// Mitsubishi GX Works2 project: SmartFarmModbusTempDx   PLC: FX3U/FX3UC

PROGRAM MAIN
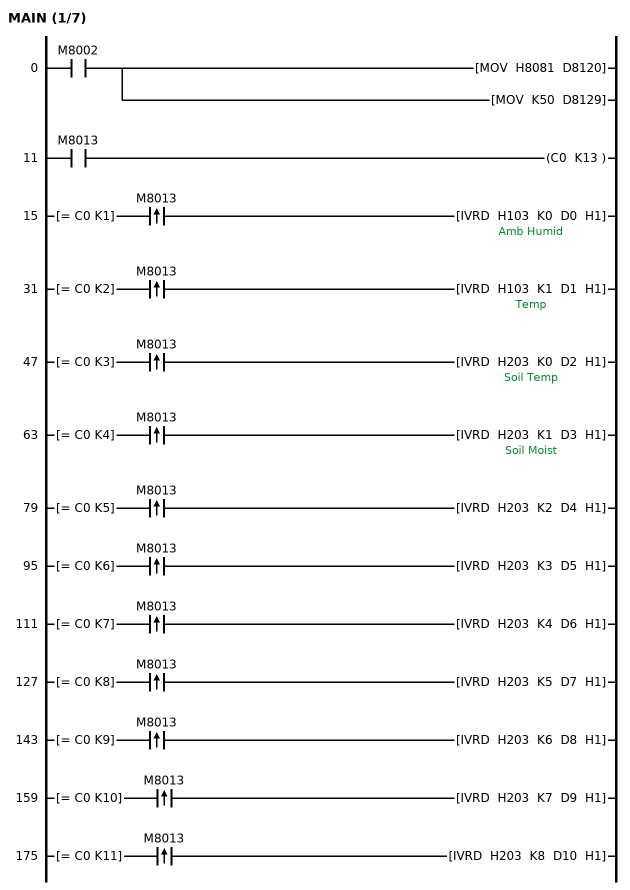
0     LD      M8002
      MOV     H8081 D8120
      MOV     K50 D8129
11    LD      M8013
      OUT     C0 K13
15    LD=     C0 K1
      ANDP    M8013
      IVRD    H103 K0 D0 H1  ; Amb Humid
31    LD=     C0 K2
      ANDP    M8013
      IVRD    H103 K1 D1 H1  ; Temp
47    LD=     C0 K3
      ANDP    M8013
      IVRD    H203 K0 D2 H1  ; Soil Temp
63    LD=     C0 K4
      ANDP    M8013
      IVRD    H203 K1 D3 H1  ; Soil Moist
79    LD=     C0 K5
      ANDP    M8013
      IVRD    H203 K2 D4 H1
95    LD=     C0 K6
      ANDP    M8013
      IVRD    H203 K3 D5 H1
111   LD=     C0 K7
      ANDP    M8013
      IVRD    H203 K4 D6 H1
127   LD=     C0 K8
      ANDP    M8013
      IVRD    H203 K5 D7 H1
143   LD=     C0 K9
      ANDP    M8013
      IVRD    H203 K6 D8 H1
159   LD=     C0 K10
      ANDP    M8013
      IVRD    H203 K7 D9 H1
175   LD=     C0 K11
      ANDP    M8013
      IVRD    H203 K8 D10 H1
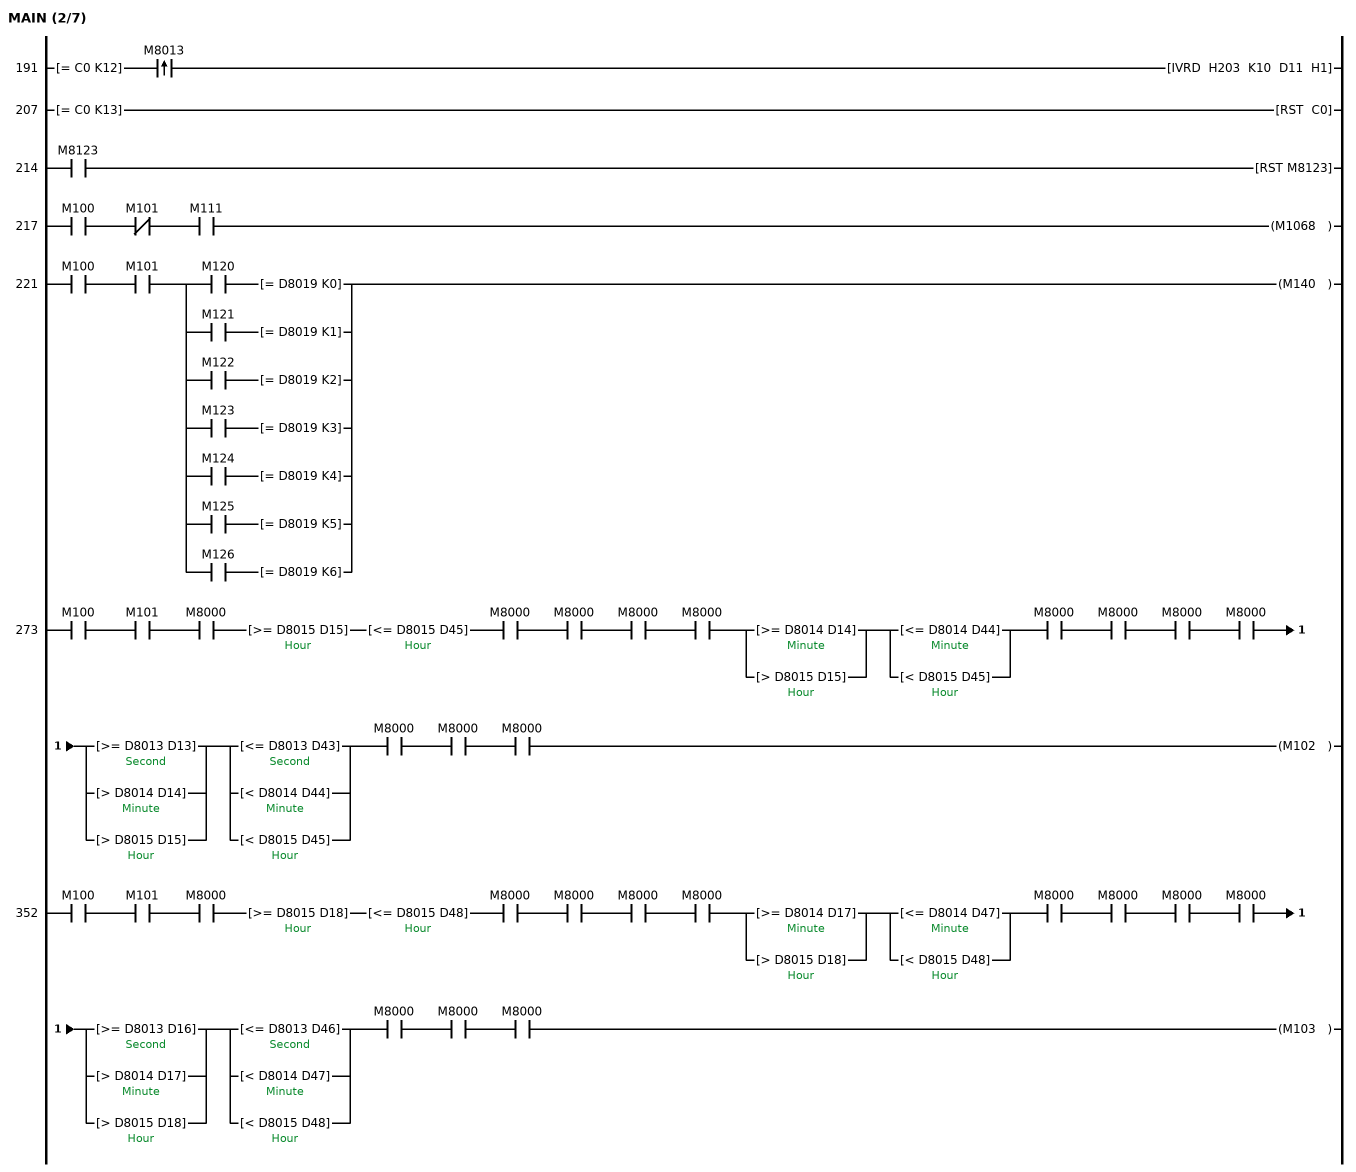
191   LD=     C0 K12
      ANDP    M8013
      IVRD    H203 K10 D11 H1
207   LD=     C0 K13
      RST     C0
214   LD      M8123
      RST     M8123
217   LD      M100
      ANI     M101
      AND     M111
      OUT     M1068
221   LD      M100
      AND     M101
      LD      M120
      AND=    D8019 K0
      LD      M121
      AND=    D8019 K1
      ORB
      LD      M122
      AND=    D8019 K2
      ORB
      LD      M123
      AND=    D8019 K3
      ORB
      LD      M124
      AND=    D8019 K4
      ORB
      LD      M125
      AND=    D8019 K5
      ORB
      LD      M126
      AND=    D8019 K6
      ORB
      ANB
      OUT     M140
273   LD      M100
      AND     M101
      AND     M8000
      AND>=   D8015 D15  ; Hour
      AND<=   D8015 D45  ; Hour
      AND     M8000
      AND     M8000
      AND     M8000
      AND     M8000
      LD>=    D8014 D14  ; Minute
      OR>     D8015 D15  ; Hour
      ANB
      LD<=    D8014 D44  ; Minute
      OR<     D8015 D45  ; Hour
      ANB
      AND     M8000
      AND     M8000
      AND     M8000
      AND     M8000
      LD>=    D8013 D13  ; Second
      OR>     D8014 D14  ; Minute
      OR>     D8015 D15  ; Hour
      ANB
      LD<=    D8013 D43  ; Second
      OR<     D8014 D44  ; Minute
      OR<     D8015 D45  ; Hour
      ANB
      AND     M8000
      AND     M8000
      AND     M8000
      OUT     M102
352   LD      M100
      AND     M101
      AND     M8000
      AND>=   D8015 D18  ; Hour
      AND<=   D8015 D48  ; Hour
      AND     M8000
      AND     M8000
      AND     M8000
      AND     M8000
      LD>=    D8014 D17  ; Minute
      OR>     D8015 D18  ; Hour
      ANB
      LD<=    D8014 D47  ; Minute
      OR<     D8015 D48  ; Hour
      ANB
      AND     M8000
      AND     M8000
      AND     M8000
      AND     M8000
      LD>=    D8013 D16  ; Second
      OR>     D8014 D17  ; Minute
      OR>     D8015 D18  ; Hour
      ANB
      LD<=    D8013 D46  ; Second
      OR<     D8014 D47  ; Minute
      OR<     D8015 D48  ; Hour
      ANB
      AND     M8000
      AND     M8000
      AND     M8000
      OUT     M103
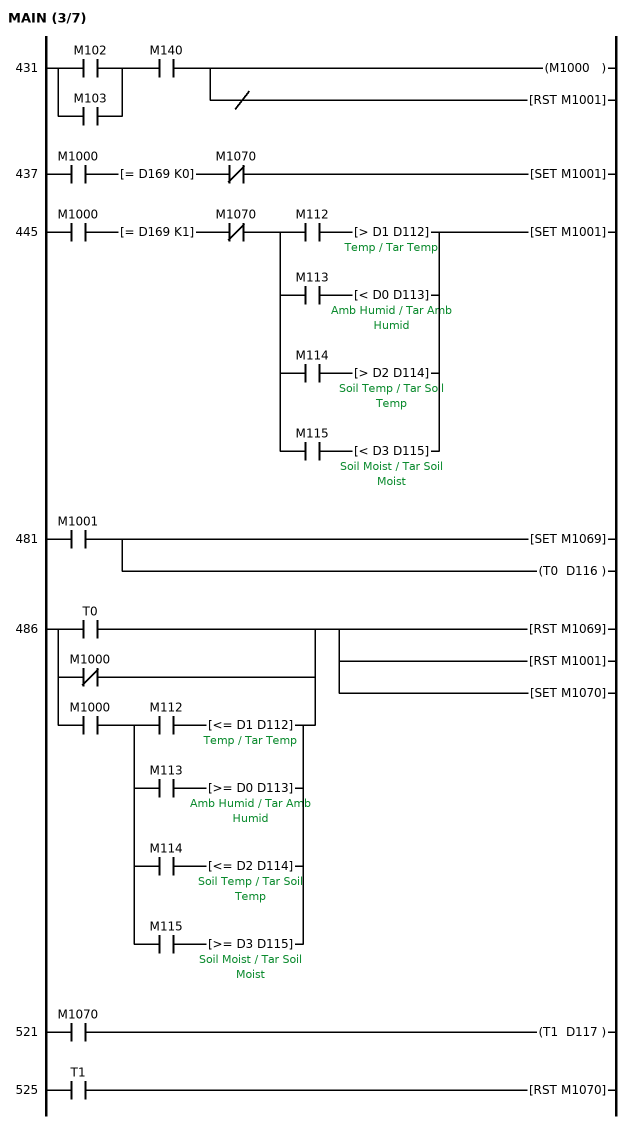
431   LD      M102
      OR      M103
      AND     M140
      OUT     M1000
      INV
      RST     M1001
437   LD      M1000
      AND=    D169 K0
      ANI     M1070
      SET     M1001
445   LD      M1000
      AND=    D169 K1
      ANI     M1070
      LD      M112
      AND>    D1 D112  ; Temp / Tar Temp
      LD      M113
      AND<    D0 D113  ; Amb Humid / Tar Amb Humid
      ORB
      LD      M114
      AND>    D2 D114  ; Soil Temp / Tar Soil Temp
      ORB
      LD      M115
      AND<    D3 D115  ; Soil Moist / Tar Soil Moist
      ORB
      ANB
      SET     M1001
481   LD      M1001
      SET     M1069
      OUT     T0 D116
486   LD      T0
      ORI     M1000
      LD      M1000
      LD      M112
      AND<=   D1 D112  ; Temp / Tar Temp
      LD      M113
      AND>=   D0 D113  ; Amb Humid / Tar Amb Humid
      ORB
      LD      M114
      AND<=   D2 D114  ; Soil Temp / Tar Soil Temp
      ORB
      LD      M115
      AND>=   D3 D115  ; Soil Moist / Tar Soil Moist
      ORB
      ANB
      ORB
      RST     M1069
      RST     M1001
      SET     M1070
521   LD      M1070
      OUT     T1 D117
525   LD      T1
      RST     M1070
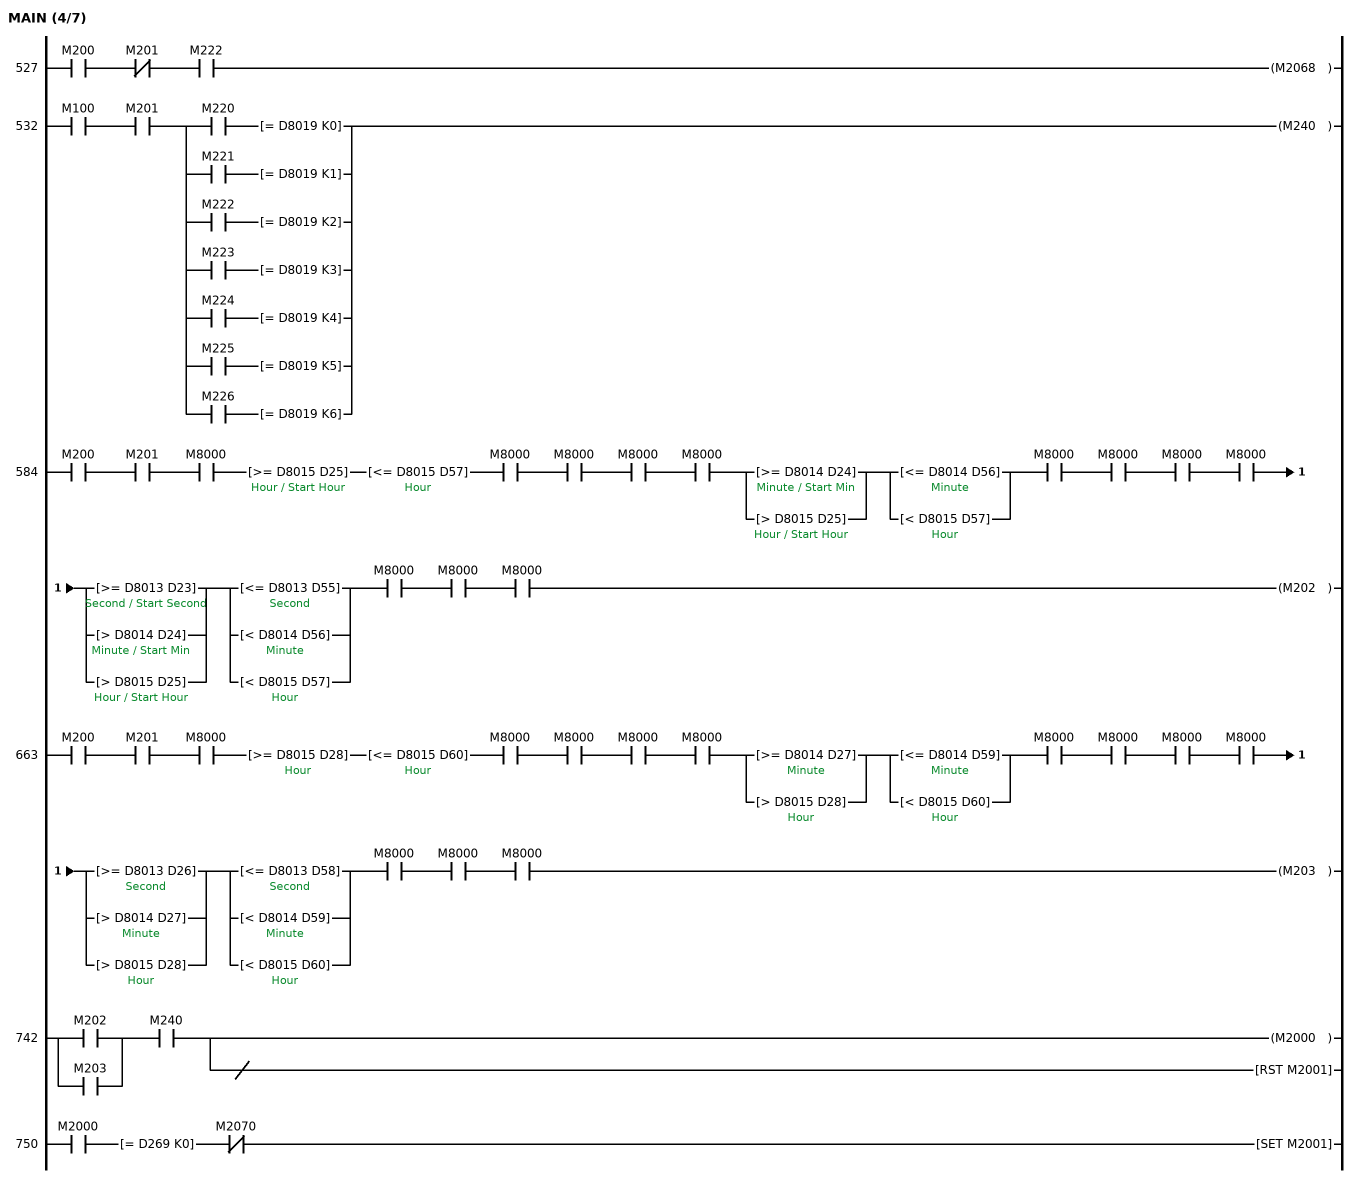
527   LD      M200
      ANI     M201
      AND     M222
      OUT     M2068
532   LD      M100
      AND     M201
      LD      M220
      AND=    D8019 K0
      LD      M221
      AND=    D8019 K1
      ORB
      LD      M222
      AND=    D8019 K2
      ORB
      LD      M223
      AND=    D8019 K3
      ORB
      LD      M224
      AND=    D8019 K4
      ORB
      LD      M225
      AND=    D8019 K5
      ORB
      LD      M226
      AND=    D8019 K6
      ORB
      ANB
      OUT     M240
584   LD      M200
      AND     M201
      AND     M8000
      AND>=   D8015 D25  ; Hour / Start Hour
      AND<=   D8015 D57  ; Hour
      AND     M8000
      AND     M8000
      AND     M8000
      AND     M8000
      LD>=    D8014 D24  ; Minute / Start Min
      OR>     D8015 D25  ; Hour / Start Hour
      ANB
      LD<=    D8014 D56  ; Minute
      OR<     D8015 D57  ; Hour
      ANB
      AND     M8000
      AND     M8000
      AND     M8000
      AND     M8000
      LD>=    D8013 D23  ; Second / Start Second
      OR>     D8014 D24  ; Minute / Start Min
      OR>     D8015 D25  ; Hour / Start Hour
      ANB
      LD<=    D8013 D55  ; Second
      OR<     D8014 D56  ; Minute
      OR<     D8015 D57  ; Hour
      ANB
      AND     M8000
      AND     M8000
      AND     M8000
      OUT     M202
663   LD      M200
      AND     M201
      AND     M8000
      AND>=   D8015 D28  ; Hour
      AND<=   D8015 D60  ; Hour
      AND     M8000
      AND     M8000
      AND     M8000
      AND     M8000
      LD>=    D8014 D27  ; Minute
      OR>     D8015 D28  ; Hour
      ANB
      LD<=    D8014 D59  ; Minute
      OR<     D8015 D60  ; Hour
      ANB
      AND     M8000
      AND     M8000
      AND     M8000
      AND     M8000
      LD>=    D8013 D26  ; Second
      OR>     D8014 D27  ; Minute
      OR>     D8015 D28  ; Hour
      ANB
      LD<=    D8013 D58  ; Second
      OR<     D8014 D59  ; Minute
      OR<     D8015 D60  ; Hour
      ANB
      AND     M8000
      AND     M8000
      AND     M8000
      OUT     M203
742   LD      M202
      OR      M203
      AND     M240
      OUT     M2000
      INV
      RST     M2001
750   LD      M2000
      AND=    D269 K0
      ANI     M2070
      SET     M2001
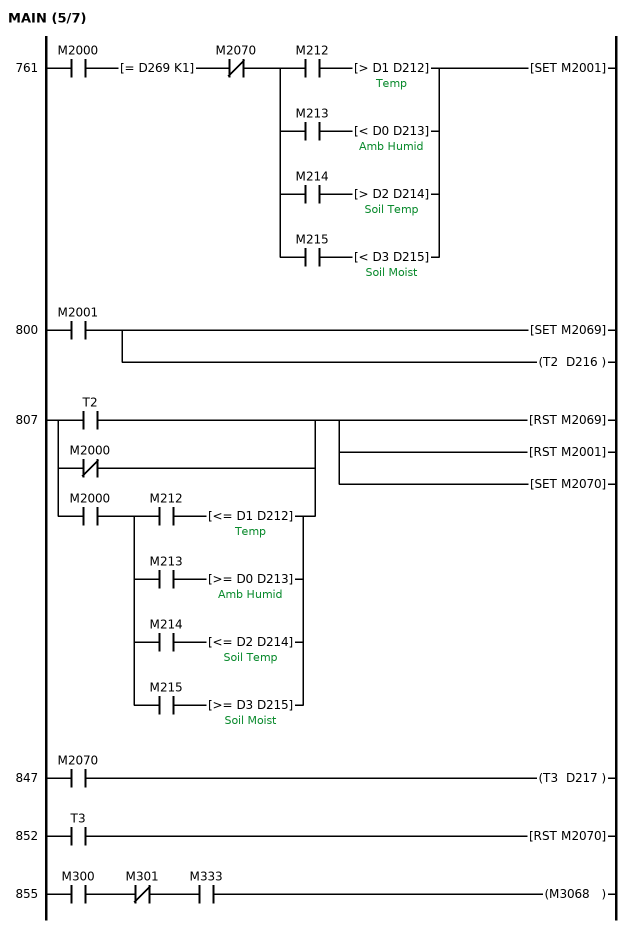
761   LD      M2000
      AND=    D269 K1
      ANI     M2070
      LD      M212
      AND>    D1 D212  ; Temp
      LD      M213
      AND<    D0 D213  ; Amb Humid
      ORB
      LD      M214
      AND>    D2 D214  ; Soil Temp
      ORB
      LD      M215
      AND<    D3 D215  ; Soil Moist
      ORB
      ANB
      SET     M2001
800   LD      M2001
      SET     M2069
      OUT     T2 D216
807   LD      T2
      ORI     M2000
      LD      M2000
      LD      M212
      AND<=   D1 D212  ; Temp
      LD      M213
      AND>=   D0 D213  ; Amb Humid
      ORB
      LD      M214
      AND<=   D2 D214  ; Soil Temp
      ORB
      LD      M215
      AND>=   D3 D215  ; Soil Moist
      ORB
      ANB
      ORB
      RST     M2069
      RST     M2001
      SET     M2070
847   LD      M2070
      OUT     T3 D217
852   LD      T3
      RST     M2070
855   LD      M300
      ANI     M301
      AND     M333
      OUT     M3068
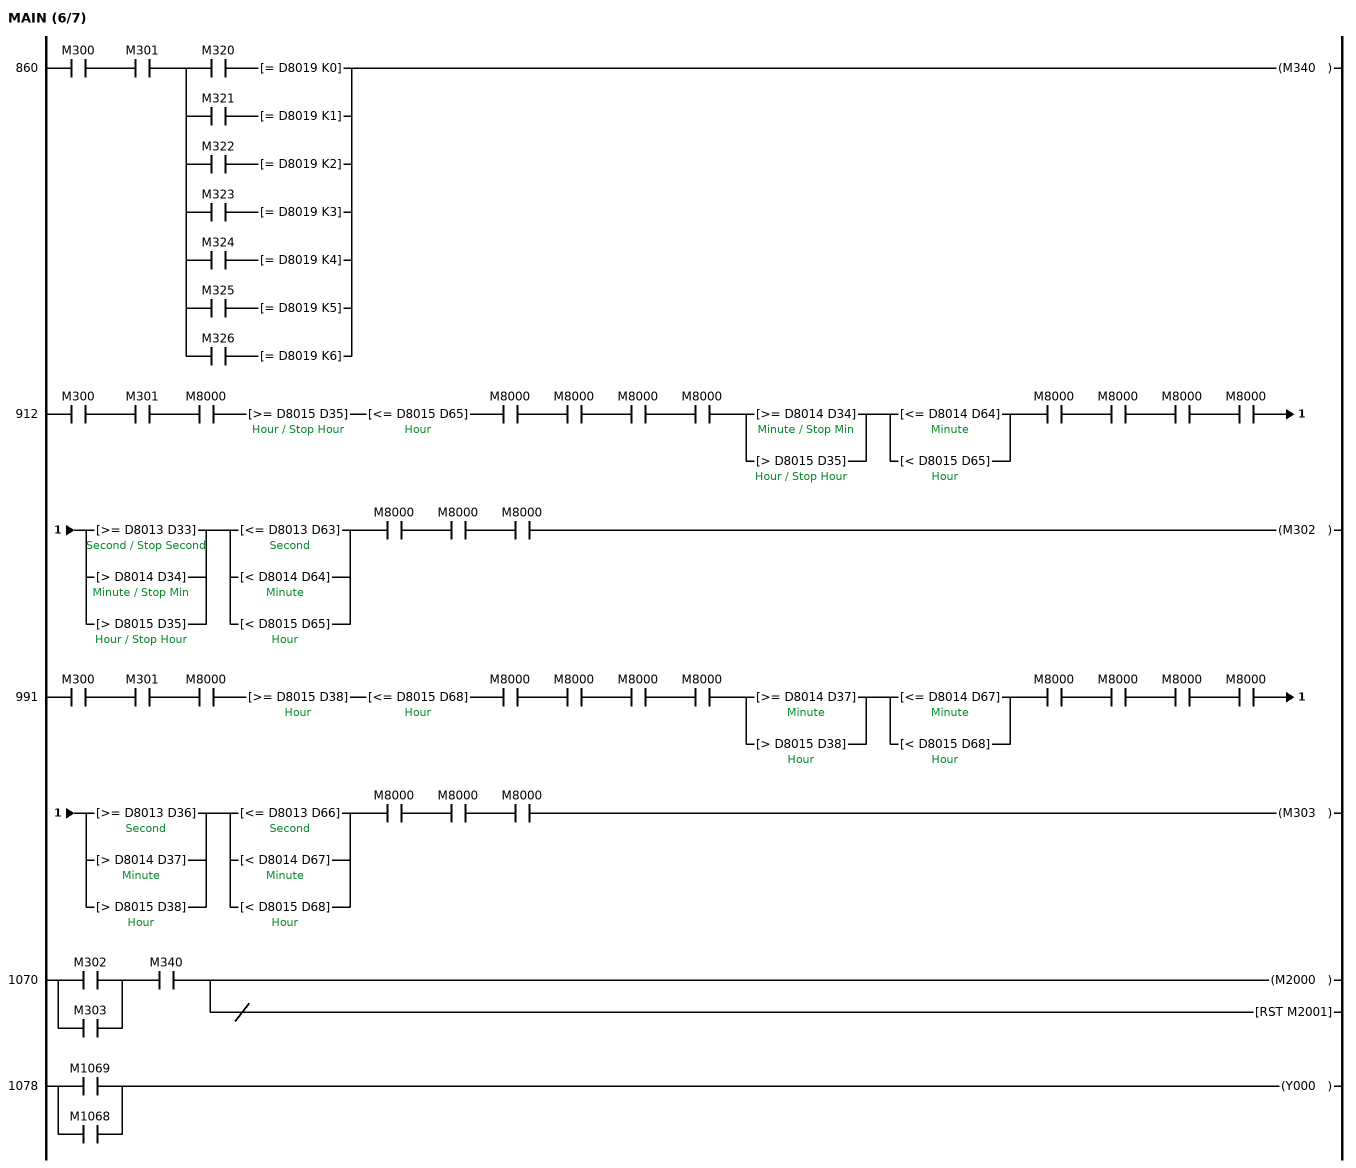
860   LD      M300
      AND     M301
      LD      M320
      AND=    D8019 K0
      LD      M321
      AND=    D8019 K1
      ORB
      LD      M322
      AND=    D8019 K2
      ORB
      LD      M323
      AND=    D8019 K3
      ORB
      LD      M324
      AND=    D8019 K4
      ORB
      LD      M325
      AND=    D8019 K5
      ORB
      LD      M326
      AND=    D8019 K6
      ORB
      ANB
      OUT     M340
912   LD      M300
      AND     M301
      AND     M8000
      AND>=   D8015 D35  ; Hour / Stop Hour
      AND<=   D8015 D65  ; Hour
      AND     M8000
      AND     M8000
      AND     M8000
      AND     M8000
      LD>=    D8014 D34  ; Minute / Stop Min
      OR>     D8015 D35  ; Hour / Stop Hour
      ANB
      LD<=    D8014 D64  ; Minute
      OR<     D8015 D65  ; Hour
      ANB
      AND     M8000
      AND     M8000
      AND     M8000
      AND     M8000
      LD>=    D8013 D33  ; Second / Stop Second
      OR>     D8014 D34  ; Minute / Stop Min
      OR>     D8015 D35  ; Hour / Stop Hour
      ANB
      LD<=    D8013 D63  ; Second
      OR<     D8014 D64  ; Minute
      OR<     D8015 D65  ; Hour
      ANB
      AND     M8000
      AND     M8000
      AND     M8000
      OUT     M302
991   LD      M300
      AND     M301
      AND     M8000
      AND>=   D8015 D38  ; Hour
      AND<=   D8015 D68  ; Hour
      AND     M8000
      AND     M8000
      AND     M8000
      AND     M8000
      LD>=    D8014 D37  ; Minute
      OR>     D8015 D38  ; Hour
      ANB
      LD<=    D8014 D67  ; Minute
      OR<     D8015 D68  ; Hour
      ANB
      AND     M8000
      AND     M8000
      AND     M8000
      AND     M8000
      LD>=    D8013 D36  ; Second
      OR>     D8014 D37  ; Minute
      OR>     D8015 D38  ; Hour
      ANB
      LD<=    D8013 D66  ; Second
      OR<     D8014 D67  ; Minute
      OR<     D8015 D68  ; Hour
      ANB
      AND     M8000
      AND     M8000
      AND     M8000
      OUT     M303
1070  LD      M302
      OR      M303
      AND     M340
      OUT     M2000
      INV
      RST     M2001
1078  LD      M1069
      OR      M1068
      OUT     Y000
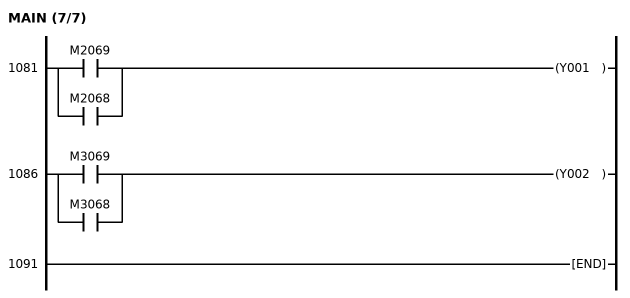
1081  LD      M2069
      OR      M2068
      OUT     Y001
1086  LD      M3069
      OR      M3068
      OUT     Y002
1091  END
END_PROGRAM
